FUNCTION_BLOCK FB_Topology
VAR_INPUT
    PLCtoIO : st_IO_Outputs; // hardware outputs
END_VAR
VAR_OUTPUT
	IOtoPLC : st_IO_Inputs; // hardware inputs
END_VAR
VAR
END_VAR

// monitor IO

METHOD HandleInputs : BOOL
VAR_INPUT
END_VAR
// ============ Hydrualic System ============

// Pressure Transducer
IOtoPLC.pressureTransducer.value := GVL_iXlinker.E_Bus.Term_1_EK1100.Term_2_EL3024.AI_Standard_Channel_1.Value;


// Proportional Valve


// Robot
IOtoPLC.robot.fault := GVL_iXlinker.E_Bus.X001_KRC4_secondary_EL6695_1001.Module_3_Default_IO.Std_In_4_Bytes.Input_DWORD_0.0;
END_METHOD

METHOD HandleOutputs : BOOL
VAR_INPUT
END_VAR
// Robot
GVL_iXlinker.E_Bus.X001_KRC4_secondary_EL6695_1001.Module_3_Default_IO.Std_Out_4_Bytes.Output_DWORD_0.0 := PLCtoIO.robot.fault;

// Pump
GVL_iXlinker.E_Bus.Term_1_EK1100.Term_3_EL2634.Channel_1.Output := PLCtoIO.hydroPump.On;
END_METHOD

END_FUNCTION_BLOCK

(* stored: Version 1.1.0.1, ProductVersion 3.1.4024.9
   POU FB_Topology: Id {d48ab407-8d9b-49c4-845c-3dec913e9feb}, SpecialFunc None
   Method HandleInputs: Id {244df69a-9a92-4686-a02a-1bd2d6abbee5}
   Method HandleOutputs: Id {916f8403-9a6a-4b2b-ae86-1fd7e0f2a6e8} *)
